DATA_BLOCK "FB_ControlRecipes_DB"
{ S7_Optimized_Access := 'TRUE' }
VERSION : 0.1
NON_RETAIN
"FB_ControlRecipes"

BEGIN

END_DATA_BLOCK

